INTERFACE I_Tagged EXTENDS Domains.I_Component

PROPERTY Tag : I_Tag
GET
END_GET
END_PROPERTY

END_INTERFACE

(* stored: Version 1.1.0.1
   Itf I_Tagged: Id {b58edee9-4fde-44ef-8cdc-e705919fec86}
   Property Tag: Id {44276dfe-612b-4762-b855-7fa4243cc2ba}
   Get Get: Id {90182557-be94-4a95-8ef7-fb2e3a0691ff} *)
